PROGRAM PRG_VLS_VACUUM
VAR
	stPTM : ST_PfeifferControl;
	fbPTM : FB_PTM_Pfeiffer;
END_VAR
VAR_INPUT
	bVLS_Ext_Press : BOOL := FALSE; // external interlock bit for window control
END_VAR

// VLS Vacuum Logic
PRG_VLS_WINDOW(bExtPress := bVLS_Ext_Press); // run the vacuum program with interlock bit

// VLS Pump
PRG_PUMP();

END_PROGRAM

(* stored: Version 1.1.0.1, ProductVersion 3.1.4024.2
   POU PRG_VLS_VACUUM: Id {54bbc3ff-d626-4728-80d9-398bf4fa229d}, SpecialFunc None *)
